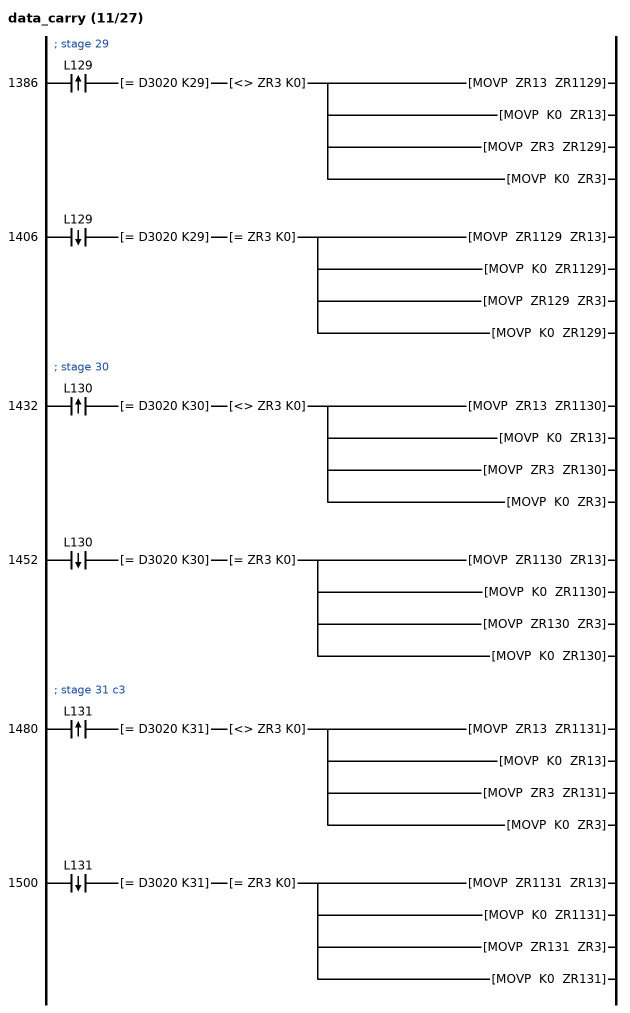
[picture p96: ladder of data_carry, rungs at steps 1386 to 1500]
; stage 29
1386  LDP     L129
      AND=    D3020 K29
      AND<>   ZR3 K0
      MOVP    ZR13 ZR1129
      MOVP    K0 ZR13
      MOVP    ZR3 ZR129
      MOVP    K0 ZR3
1406  LDF     L129
      AND=    D3020 K29
      AND=    ZR3 K0
      MOVP    ZR1129 ZR13
      MOVP    K0 ZR1129
      MOVP    ZR129 ZR3
      MOVP    K0 ZR129
; stage 30
1432  LDP     L130
      AND=    D3020 K30
      AND<>   ZR3 K0
      MOVP    ZR13 ZR1130
      MOVP    K0 ZR13
      MOVP    ZR3 ZR130
      MOVP    K0 ZR3
1452  LDF     L130
      AND=    D3020 K30
      AND=    ZR3 K0
      MOVP    ZR1130 ZR13
      MOVP    K0 ZR1130
      MOVP    ZR130 ZR3
      MOVP    K0 ZR130
; stage 31 c3
1480  LDP     L131
      AND=    D3020 K31
      AND<>   ZR3 K0
      MOVP    ZR13 ZR1131
      MOVP    K0 ZR13
      MOVP    ZR3 ZR131
      MOVP    K0 ZR3
1500  LDF     L131
      AND=    D3020 K31
      AND=    ZR3 K0
      MOVP    ZR1131 ZR13
      MOVP    K0 ZR1131
      MOVP    ZR131 ZR3
      MOVP    K0 ZR131
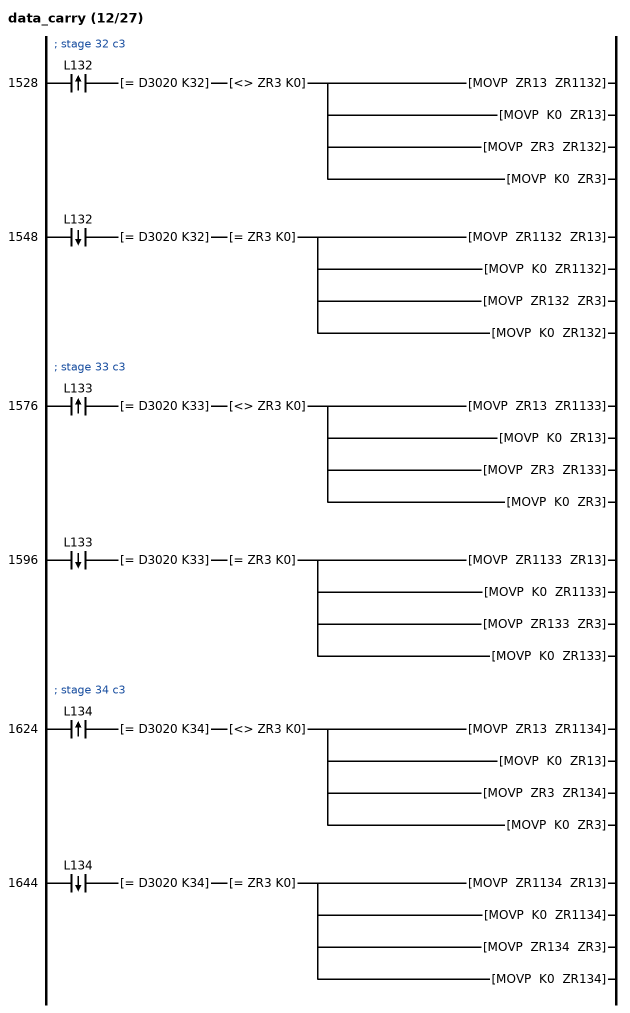
; stage 32 c3
1528  LDP     L132
      AND=    D3020 K32
      AND<>   ZR3 K0
      MOVP    ZR13 ZR1132
      MOVP    K0 ZR13
      MOVP    ZR3 ZR132
      MOVP    K0 ZR3
1548  LDF     L132
      AND=    D3020 K32
      AND=    ZR3 K0
      MOVP    ZR1132 ZR13
      MOVP    K0 ZR1132
      MOVP    ZR132 ZR3
      MOVP    K0 ZR132
; stage 33 c3
1576  LDP     L133
      AND=    D3020 K33
      AND<>   ZR3 K0
      MOVP    ZR13 ZR1133
      MOVP    K0 ZR13
      MOVP    ZR3 ZR133
      MOVP    K0 ZR3
1596  LDF     L133
      AND=    D3020 K33
      AND=    ZR3 K0
      MOVP    ZR1133 ZR13
      MOVP    K0 ZR1133
      MOVP    ZR133 ZR3
      MOVP    K0 ZR133
; stage 34 c3
1624  LDP     L134
      AND=    D3020 K34
      AND<>   ZR3 K0
      MOVP    ZR13 ZR1134
      MOVP    K0 ZR13
      MOVP    ZR3 ZR134
      MOVP    K0 ZR3
1644  LDF     L134
      AND=    D3020 K34
      AND=    ZR3 K0
      MOVP    ZR1134 ZR13
      MOVP    K0 ZR1134
      MOVP    ZR134 ZR3
      MOVP    K0 ZR134
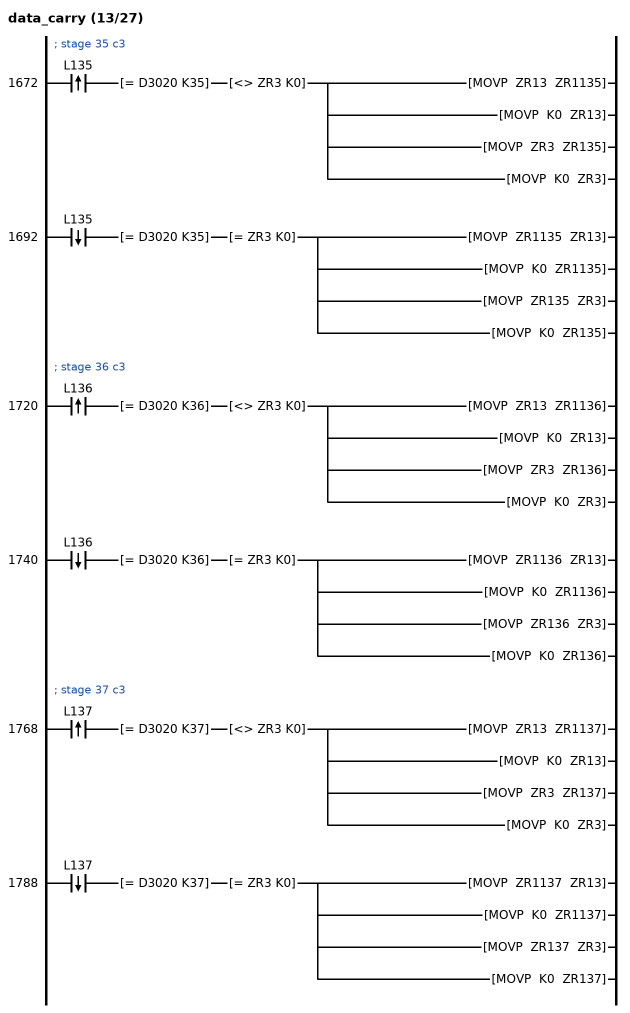
; stage 35 c3
1672  LDP     L135
      AND=    D3020 K35
      AND<>   ZR3 K0
      MOVP    ZR13 ZR1135
      MOVP    K0 ZR13
      MOVP    ZR3 ZR135
      MOVP    K0 ZR3
1692  LDF     L135
      AND=    D3020 K35
      AND=    ZR3 K0
      MOVP    ZR1135 ZR13
      MOVP    K0 ZR1135
      MOVP    ZR135 ZR3
      MOVP    K0 ZR135
; stage 36 c3
1720  LDP     L136
      AND=    D3020 K36
      AND<>   ZR3 K0
      MOVP    ZR13 ZR1136
      MOVP    K0 ZR13
      MOVP    ZR3 ZR136
      MOVP    K0 ZR3
1740  LDF     L136
      AND=    D3020 K36
      AND=    ZR3 K0
      MOVP    ZR1136 ZR13
      MOVP    K0 ZR1136
      MOVP    ZR136 ZR3
      MOVP    K0 ZR136
; stage 37 c3
1768  LDP     L137
      AND=    D3020 K37
      AND<>   ZR3 K0
      MOVP    ZR13 ZR1137
      MOVP    K0 ZR13
      MOVP    ZR3 ZR137
      MOVP    K0 ZR3
1788  LDF     L137
      AND=    D3020 K37
      AND=    ZR3 K0
      MOVP    ZR1137 ZR13
      MOVP    K0 ZR1137
      MOVP    ZR137 ZR3
      MOVP    K0 ZR137
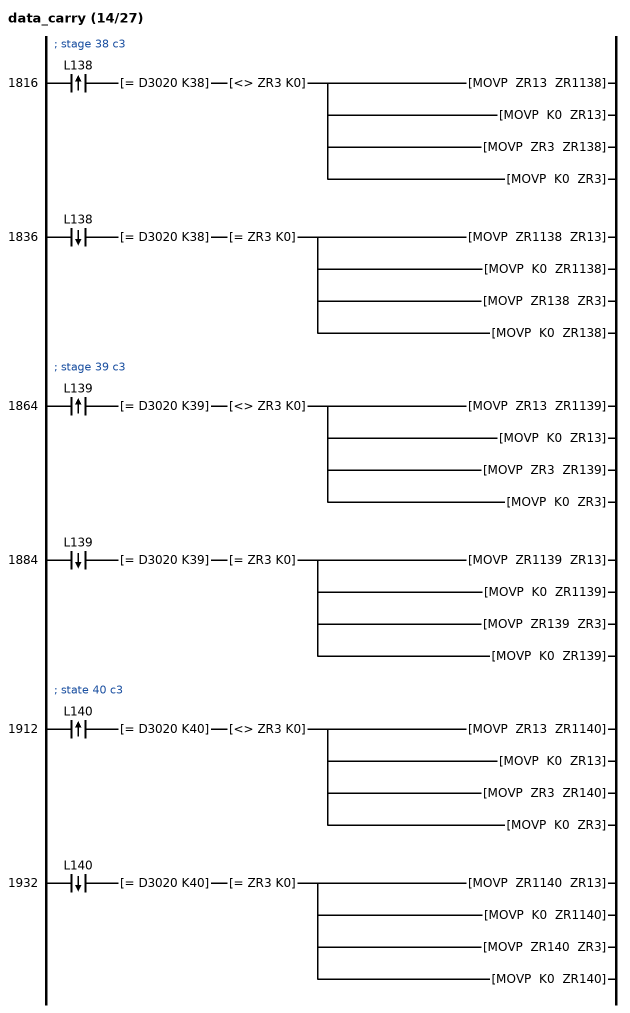
; stage 38 c3
1816  LDP     L138
      AND=    D3020 K38
      AND<>   ZR3 K0
      MOVP    ZR13 ZR1138
      MOVP    K0 ZR13
      MOVP    ZR3 ZR138
      MOVP    K0 ZR3
1836  LDF     L138
      AND=    D3020 K38
      AND=    ZR3 K0
      MOVP    ZR1138 ZR13
      MOVP    K0 ZR1138
      MOVP    ZR138 ZR3
      MOVP    K0 ZR138
; stage 39 c3
1864  LDP     L139
      AND=    D3020 K39
      AND<>   ZR3 K0
      MOVP    ZR13 ZR1139
      MOVP    K0 ZR13
      MOVP    ZR3 ZR139
      MOVP    K0 ZR3
1884  LDF     L139
      AND=    D3020 K39
      AND=    ZR3 K0
      MOVP    ZR1139 ZR13
      MOVP    K0 ZR1139
      MOVP    ZR139 ZR3
      MOVP    K0 ZR139
; state 40 c3
1912  LDP     L140
      AND=    D3020 K40
      AND<>   ZR3 K0
      MOVP    ZR13 ZR1140
      MOVP    K0 ZR13
      MOVP    ZR3 ZR140
      MOVP    K0 ZR3
1932  LDF     L140
      AND=    D3020 K40
      AND=    ZR3 K0
      MOVP    ZR1140 ZR13
      MOVP    K0 ZR1140
      MOVP    ZR140 ZR3
      MOVP    K0 ZR140
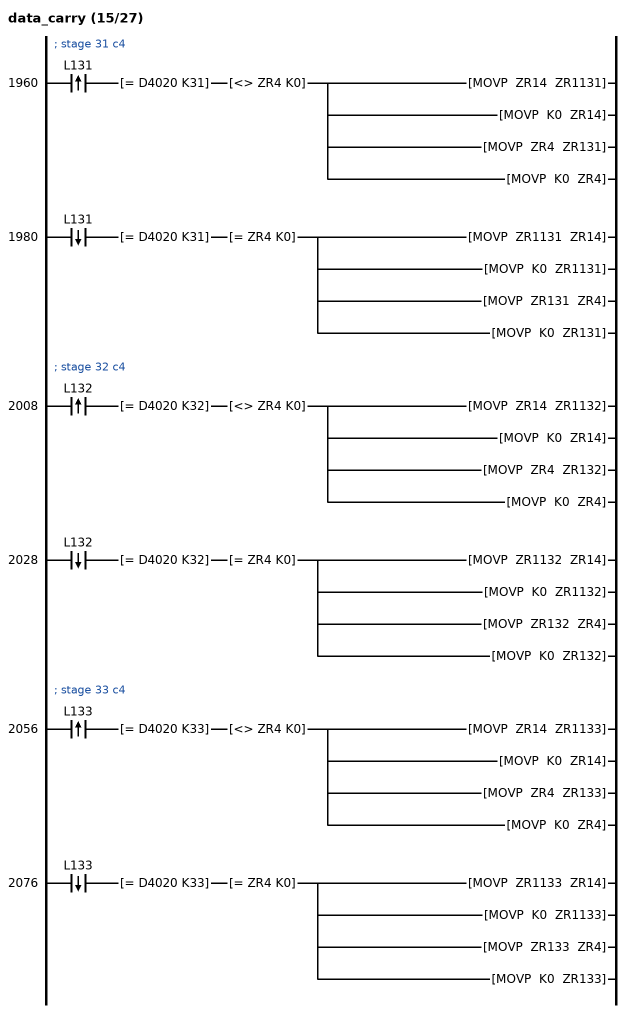
; stage 31 c4
1960  LDP     L131
      AND=    D4020 K31
      AND<>   ZR4 K0
      MOVP    ZR14 ZR1131
      MOVP    K0 ZR14
      MOVP    ZR4 ZR131
      MOVP    K0 ZR4
1980  LDF     L131
      AND=    D4020 K31
      AND=    ZR4 K0
      MOVP    ZR1131 ZR14
      MOVP    K0 ZR1131
      MOVP    ZR131 ZR4
      MOVP    K0 ZR131
; stage 32 c4
2008  LDP     L132
      AND=    D4020 K32
      AND<>   ZR4 K0
      MOVP    ZR14 ZR1132
      MOVP    K0 ZR14
      MOVP    ZR4 ZR132
      MOVP    K0 ZR4
2028  LDF     L132
      AND=    D4020 K32
      AND=    ZR4 K0
      MOVP    ZR1132 ZR14
      MOVP    K0 ZR1132
      MOVP    ZR132 ZR4
      MOVP    K0 ZR132
; stage 33 c4
2056  LDP     L133
      AND=    D4020 K33
      AND<>   ZR4 K0
      MOVP    ZR14 ZR1133
      MOVP    K0 ZR14
      MOVP    ZR4 ZR133
      MOVP    K0 ZR4
2076  LDF     L133
      AND=    D4020 K33
      AND=    ZR4 K0
      MOVP    ZR1133 ZR14
      MOVP    K0 ZR1133
      MOVP    ZR133 ZR4
      MOVP    K0 ZR133
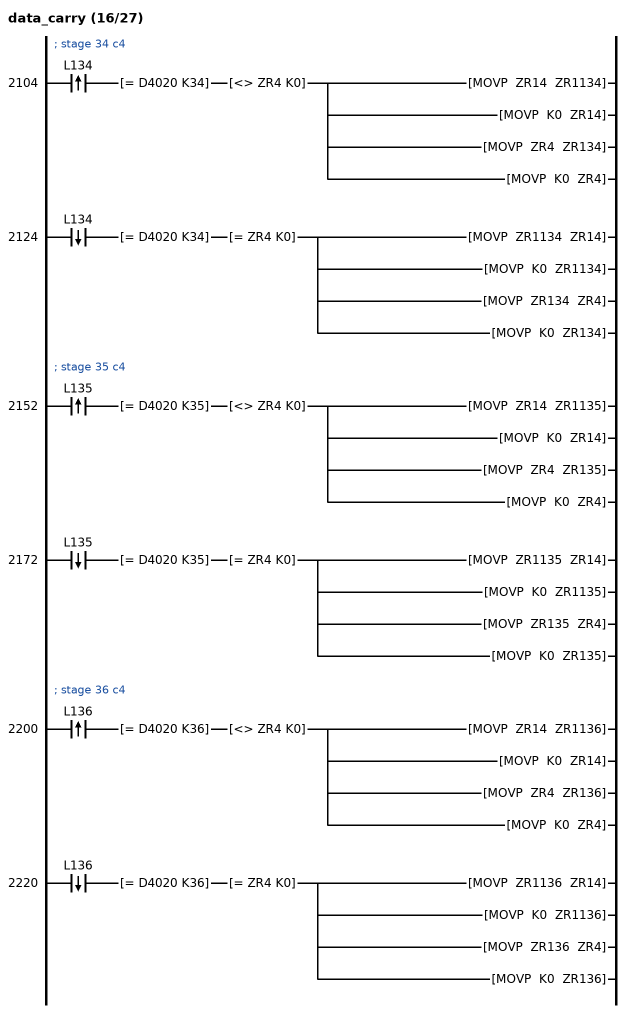
; stage 34 c4
2104  LDP     L134
      AND=    D4020 K34
      AND<>   ZR4 K0
      MOVP    ZR14 ZR1134
      MOVP    K0 ZR14
      MOVP    ZR4 ZR134
      MOVP    K0 ZR4
2124  LDF     L134
      AND=    D4020 K34
      AND=    ZR4 K0
      MOVP    ZR1134 ZR14
      MOVP    K0 ZR1134
      MOVP    ZR134 ZR4
      MOVP    K0 ZR134
; stage 35 c4
2152  LDP     L135
      AND=    D4020 K35
      AND<>   ZR4 K0
      MOVP    ZR14 ZR1135
      MOVP    K0 ZR14
      MOVP    ZR4 ZR135
      MOVP    K0 ZR4
2172  LDF     L135
      AND=    D4020 K35
      AND=    ZR4 K0
      MOVP    ZR1135 ZR14
      MOVP    K0 ZR1135
      MOVP    ZR135 ZR4
      MOVP    K0 ZR135
; stage 36 c4
2200  LDP     L136
      AND=    D4020 K36
      AND<>   ZR4 K0
      MOVP    ZR14 ZR1136
      MOVP    K0 ZR14
      MOVP    ZR4 ZR136
      MOVP    K0 ZR4
2220  LDF     L136
      AND=    D4020 K36
      AND=    ZR4 K0
      MOVP    ZR1136 ZR14
      MOVP    K0 ZR1136
      MOVP    ZR136 ZR4
      MOVP    K0 ZR136
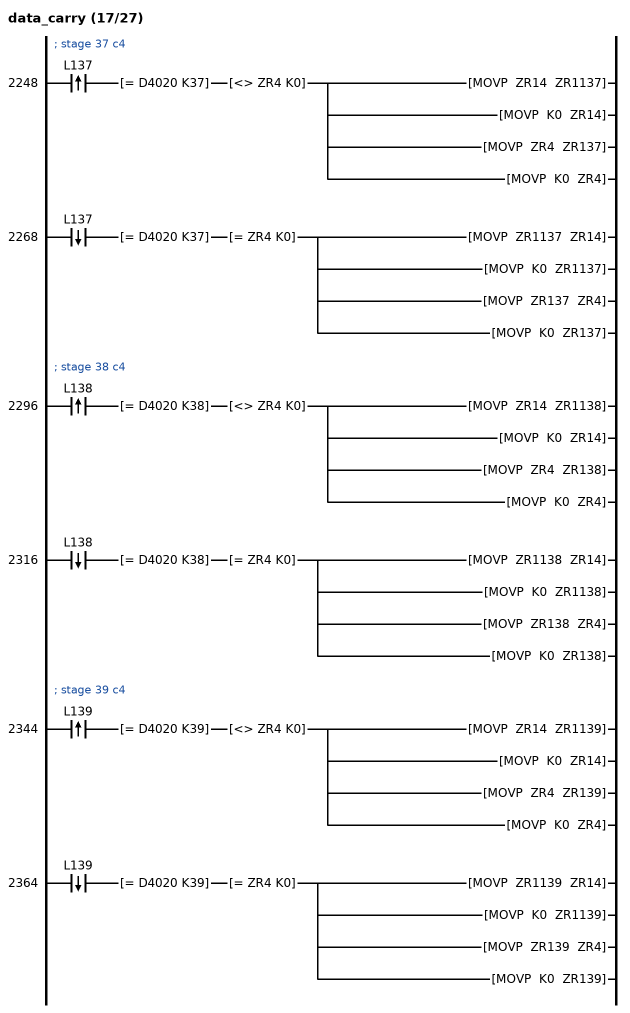
; stage 37 c4
2248  LDP     L137
      AND=    D4020 K37
      AND<>   ZR4 K0
      MOVP    ZR14 ZR1137
      MOVP    K0 ZR14
      MOVP    ZR4 ZR137
      MOVP    K0 ZR4
2268  LDF     L137
      AND=    D4020 K37
      AND=    ZR4 K0
      MOVP    ZR1137 ZR14
      MOVP    K0 ZR1137
      MOVP    ZR137 ZR4
      MOVP    K0 ZR137
; stage 38 c4
2296  LDP     L138
      AND=    D4020 K38
      AND<>   ZR4 K0
      MOVP    ZR14 ZR1138
      MOVP    K0 ZR14
      MOVP    ZR4 ZR138
      MOVP    K0 ZR4
2316  LDF     L138
      AND=    D4020 K38
      AND=    ZR4 K0
      MOVP    ZR1138 ZR14
      MOVP    K0 ZR1138
      MOVP    ZR138 ZR4
      MOVP    K0 ZR138
; stage 39 c4
2344  LDP     L139
      AND=    D4020 K39
      AND<>   ZR4 K0
      MOVP    ZR14 ZR1139
      MOVP    K0 ZR14
      MOVP    ZR4 ZR139
      MOVP    K0 ZR4
2364  LDF     L139
      AND=    D4020 K39
      AND=    ZR4 K0
      MOVP    ZR1139 ZR14
      MOVP    K0 ZR1139
      MOVP    ZR139 ZR4
      MOVP    K0 ZR139
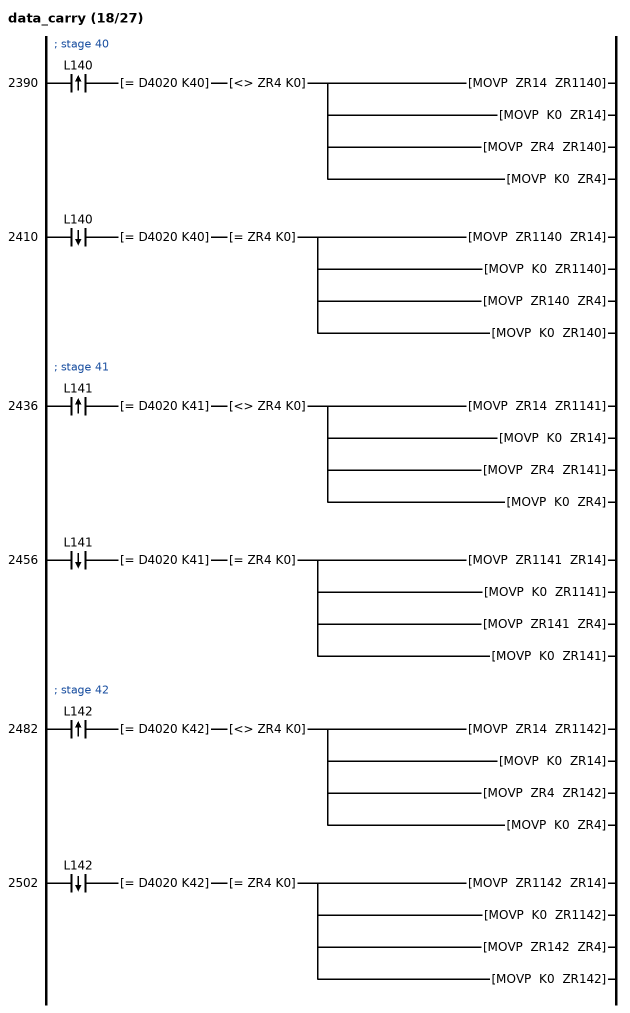
; stage 40
2390  LDP     L140
      AND=    D4020 K40
      AND<>   ZR4 K0
      MOVP    ZR14 ZR1140
      MOVP    K0 ZR14
      MOVP    ZR4 ZR140
      MOVP    K0 ZR4
2410  LDF     L140
      AND=    D4020 K40
      AND=    ZR4 K0
      MOVP    ZR1140 ZR14
      MOVP    K0 ZR1140
      MOVP    ZR140 ZR4
      MOVP    K0 ZR140
; stage 41
2436  LDP     L141
      AND=    D4020 K41
      AND<>   ZR4 K0
      MOVP    ZR14 ZR1141
      MOVP    K0 ZR14
      MOVP    ZR4 ZR141
      MOVP    K0 ZR4
2456  LDF     L141
      AND=    D4020 K41
      AND=    ZR4 K0
      MOVP    ZR1141 ZR14
      MOVP    K0 ZR1141
      MOVP    ZR141 ZR4
      MOVP    K0 ZR141
; stage 42
2482  LDP     L142
      AND=    D4020 K42
      AND<>   ZR4 K0
      MOVP    ZR14 ZR1142
      MOVP    K0 ZR14
      MOVP    ZR4 ZR142
      MOVP    K0 ZR4
2502  LDF     L142
      AND=    D4020 K42
      AND=    ZR4 K0
      MOVP    ZR1142 ZR14
      MOVP    K0 ZR1142
      MOVP    ZR142 ZR4
      MOVP    K0 ZR142
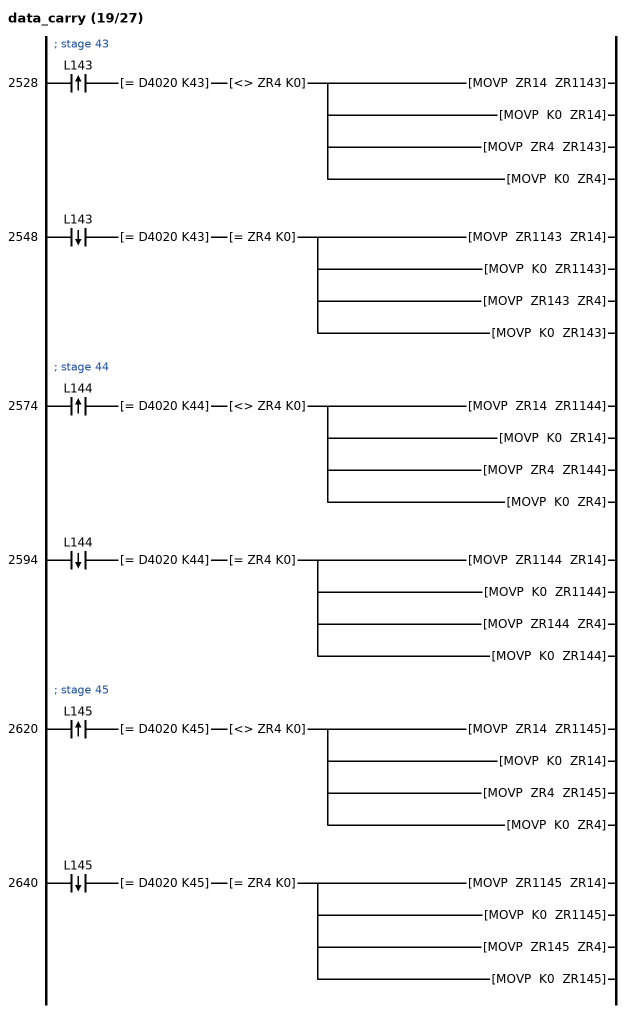
; stage 43
2528  LDP     L143
      AND=    D4020 K43
      AND<>   ZR4 K0
      MOVP    ZR14 ZR1143
      MOVP    K0 ZR14
      MOVP    ZR4 ZR143
      MOVP    K0 ZR4
2548  LDF     L143
      AND=    D4020 K43
      AND=    ZR4 K0
      MOVP    ZR1143 ZR14
      MOVP    K0 ZR1143
      MOVP    ZR143 ZR4
      MOVP    K0 ZR143
; stage 44
2574  LDP     L144
      AND=    D4020 K44
      AND<>   ZR4 K0
      MOVP    ZR14 ZR1144
      MOVP    K0 ZR14
      MOVP    ZR4 ZR144
      MOVP    K0 ZR4
2594  LDF     L144
      AND=    D4020 K44
      AND=    ZR4 K0
      MOVP    ZR1144 ZR14
      MOVP    K0 ZR1144
      MOVP    ZR144 ZR4
      MOVP    K0 ZR144
; stage 45
2620  LDP     L145
      AND=    D4020 K45
      AND<>   ZR4 K0
      MOVP    ZR14 ZR1145
      MOVP    K0 ZR14
      MOVP    ZR4 ZR145
      MOVP    K0 ZR4
2640  LDF     L145
      AND=    D4020 K45
      AND=    ZR4 K0
      MOVP    ZR1145 ZR14
      MOVP    K0 ZR1145
      MOVP    ZR145 ZR4
      MOVP    K0 ZR145
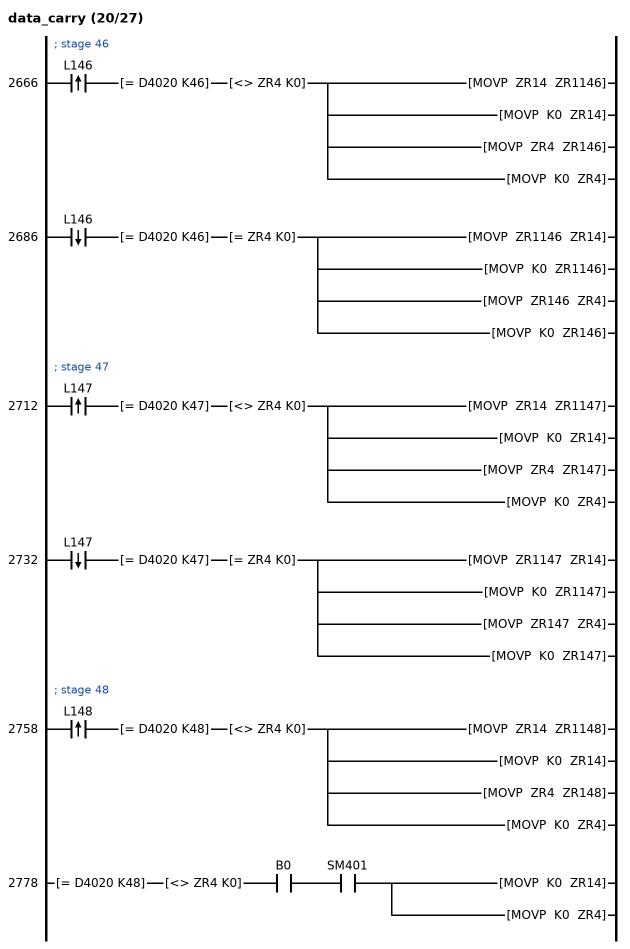
; stage 46
2666  LDP     L146
      AND=    D4020 K46
      AND<>   ZR4 K0
      MOVP    ZR14 ZR1146
      MOVP    K0 ZR14
      MOVP    ZR4 ZR146
      MOVP    K0 ZR4
2686  LDF     L146
      AND=    D4020 K46
      AND=    ZR4 K0
      MOVP    ZR1146 ZR14
      MOVP    K0 ZR1146
      MOVP    ZR146 ZR4
      MOVP    K0 ZR146
; stage 47
2712  LDP     L147
      AND=    D4020 K47
      AND<>   ZR4 K0
      MOVP    ZR14 ZR1147
      MOVP    K0 ZR14
      MOVP    ZR4 ZR147
      MOVP    K0 ZR4
2732  LDF     L147
      AND=    D4020 K47
      AND=    ZR4 K0
      MOVP    ZR1147 ZR14
      MOVP    K0 ZR1147
      MOVP    ZR147 ZR4
      MOVP    K0 ZR147
; stage 48
2758  LDP     L148
      AND=    D4020 K48
      AND<>   ZR4 K0
      MOVP    ZR14 ZR1148
      MOVP    K0 ZR14
      MOVP    ZR4 ZR148
      MOVP    K0 ZR4
2778  LD=     D4020 K48
      AND<>   ZR4 K0
      AND     B0
      AND     SM401
      MOVP    K0 ZR14
      MOVP    K0 ZR4
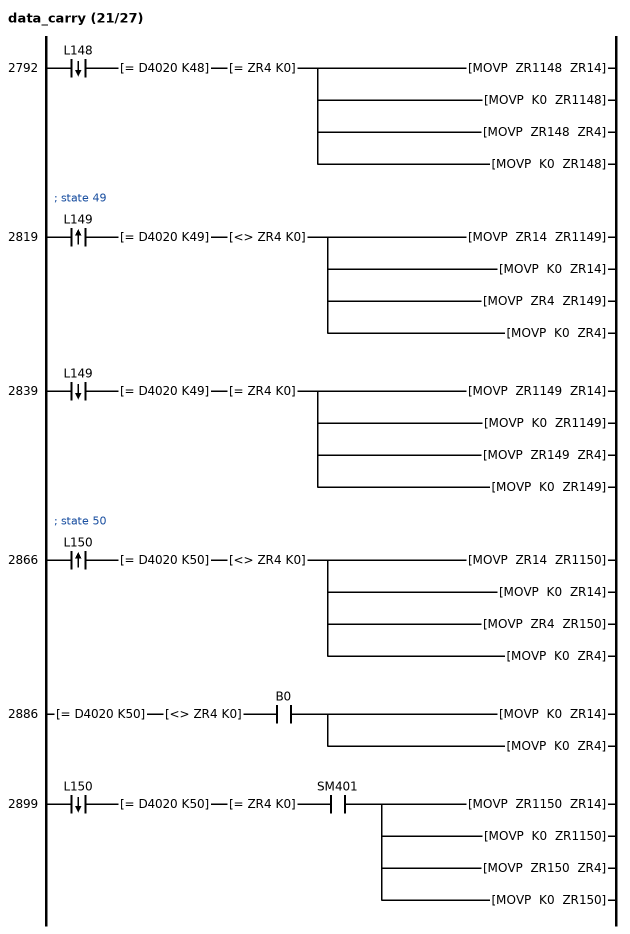
2792  LDF     L148
      AND=    D4020 K48
      AND=    ZR4 K0
      MOVP    ZR1148 ZR14
      MOVP    K0 ZR1148
      MOVP    ZR148 ZR4
      MOVP    K0 ZR148
; state 49
2819  LDP     L149
      AND=    D4020 K49
      AND<>   ZR4 K0
      MOVP    ZR14 ZR1149
      MOVP    K0 ZR14
      MOVP    ZR4 ZR149
      MOVP    K0 ZR4
2839  LDF     L149
      AND=    D4020 K49
      AND=    ZR4 K0
      MOVP    ZR1149 ZR14
      MOVP    K0 ZR1149
      MOVP    ZR149 ZR4
      MOVP    K0 ZR149
; state 50
2866  LDP     L150
      AND=    D4020 K50
      AND<>   ZR4 K0
      MOVP    ZR14 ZR1150
      MOVP    K0 ZR14
      MOVP    ZR4 ZR150
      MOVP    K0 ZR4
2886  LD=     D4020 K50
      AND<>   ZR4 K0
      AND     B0
      MOVP    K0 ZR14
      MOVP    K0 ZR4
2899  LDF     L150
      AND=    D4020 K50
      AND=    ZR4 K0
      AND     SM401
      MOVP    ZR1150 ZR14
      MOVP    K0 ZR1150
      MOVP    ZR150 ZR4
      MOVP    K0 ZR150
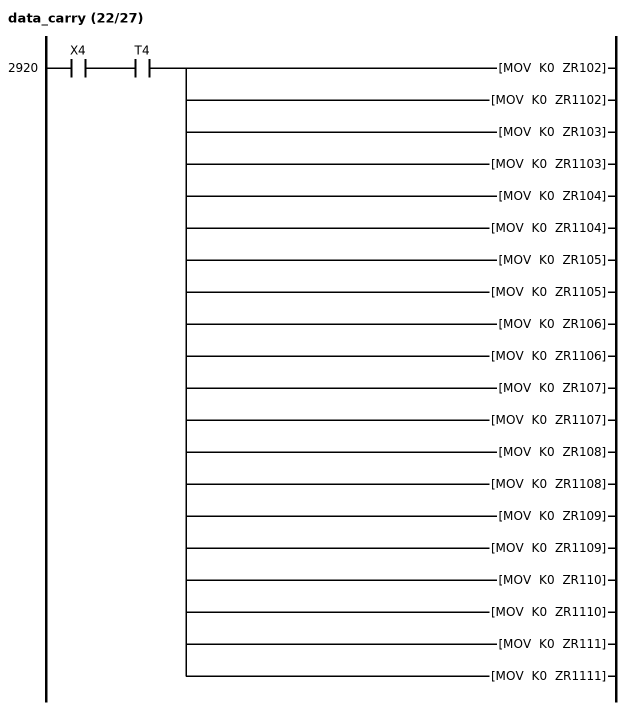
2920  LD      X4
      AND     T4
      MOV     K0 ZR102
      MOV     K0 ZR1102
      MOV     K0 ZR103
      MOV     K0 ZR1103
      MOV     K0 ZR104
      MOV     K0 ZR1104
      MOV     K0 ZR105
      MOV     K0 ZR1105
      MOV     K0 ZR106
      MOV     K0 ZR1106
      MOV     K0 ZR107
      MOV     K0 ZR1107
      MOV     K0 ZR108
      MOV     K0 ZR1108
      MOV     K0 ZR109
      MOV     K0 ZR1109
      MOV     K0 ZR110
      MOV     K0 ZR1110
      MOV     K0 ZR111
      MOV     K0 ZR1111
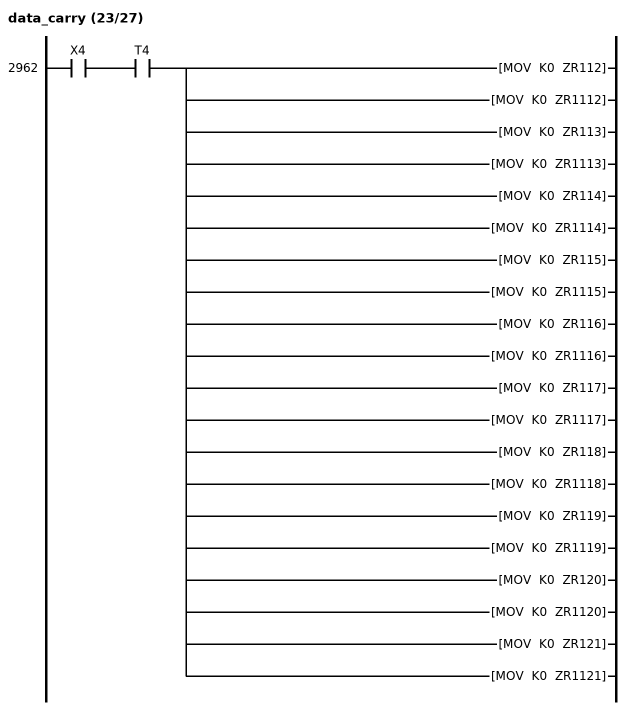
2962  LD      X4
      AND     T4
      MOV     K0 ZR112
      MOV     K0 ZR1112
      MOV     K0 ZR113
      MOV     K0 ZR1113
      MOV     K0 ZR114
      MOV     K0 ZR1114
      MOV     K0 ZR115
      MOV     K0 ZR1115
      MOV     K0 ZR116
      MOV     K0 ZR1116
      MOV     K0 ZR117
      MOV     K0 ZR1117
      MOV     K0 ZR118
      MOV     K0 ZR1118
      MOV     K0 ZR119
      MOV     K0 ZR1119
      MOV     K0 ZR120
      MOV     K0 ZR1120
      MOV     K0 ZR121
      MOV     K0 ZR1121
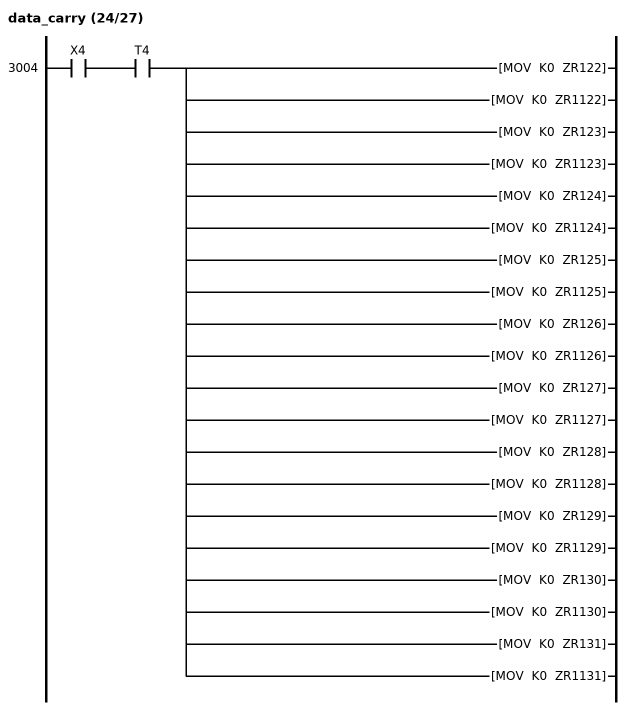
3004  LD      X4
      AND     T4
      MOV     K0 ZR122
      MOV     K0 ZR1122
      MOV     K0 ZR123
      MOV     K0 ZR1123
      MOV     K0 ZR124
      MOV     K0 ZR1124
      MOV     K0 ZR125
      MOV     K0 ZR1125
      MOV     K0 ZR126
      MOV     K0 ZR1126
      MOV     K0 ZR127
      MOV     K0 ZR1127
      MOV     K0 ZR128
      MOV     K0 ZR1128
      MOV     K0 ZR129
      MOV     K0 ZR1129
      MOV     K0 ZR130
      MOV     K0 ZR1130
      MOV     K0 ZR131
      MOV     K0 ZR1131
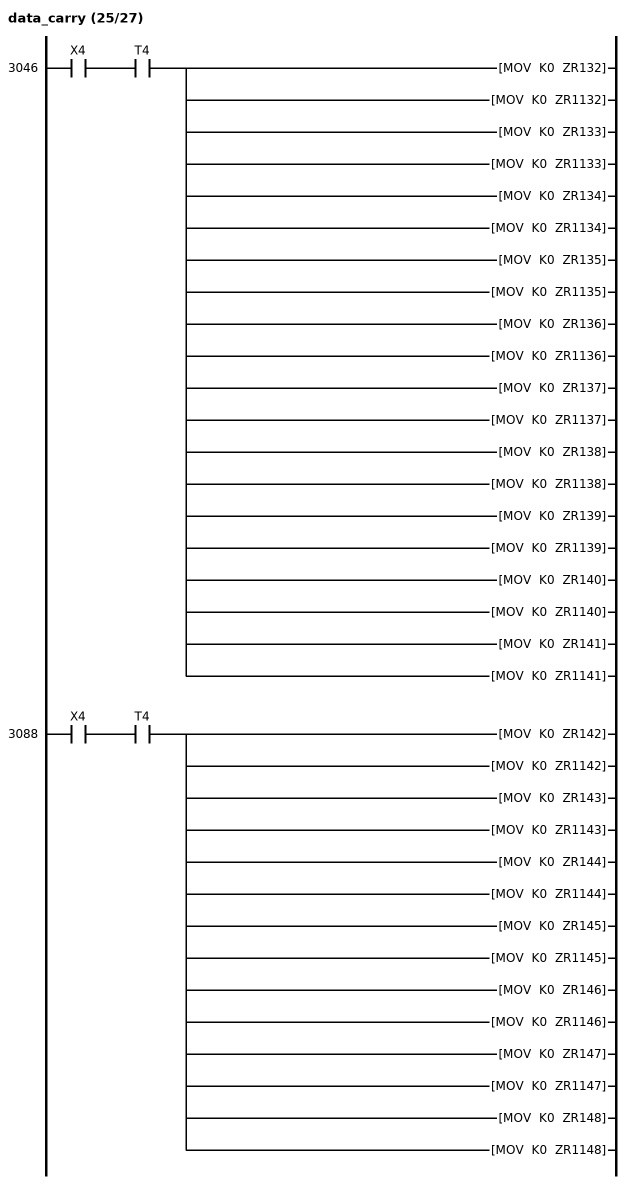
3046  LD      X4
      AND     T4
      MOV     K0 ZR132
      MOV     K0 ZR1132
      MOV     K0 ZR133
      MOV     K0 ZR1133
      MOV     K0 ZR134
      MOV     K0 ZR1134
      MOV     K0 ZR135
      MOV     K0 ZR1135
      MOV     K0 ZR136
      MOV     K0 ZR1136
      MOV     K0 ZR137
      MOV     K0 ZR1137
      MOV     K0 ZR138
      MOV     K0 ZR1138
      MOV     K0 ZR139
      MOV     K0 ZR1139
      MOV     K0 ZR140
      MOV     K0 ZR1140
      MOV     K0 ZR141
      MOV     K0 ZR1141
3088  LD      X4
      AND     T4
      MOV     K0 ZR142
      MOV     K0 ZR1142
      MOV     K0 ZR143
      MOV     K0 ZR1143
      MOV     K0 ZR144
      MOV     K0 ZR1144
      MOV     K0 ZR145
      MOV     K0 ZR1145
      MOV     K0 ZR146
      MOV     K0 ZR1146
      MOV     K0 ZR147
      MOV     K0 ZR1147
      MOV     K0 ZR148
      MOV     K0 ZR1148
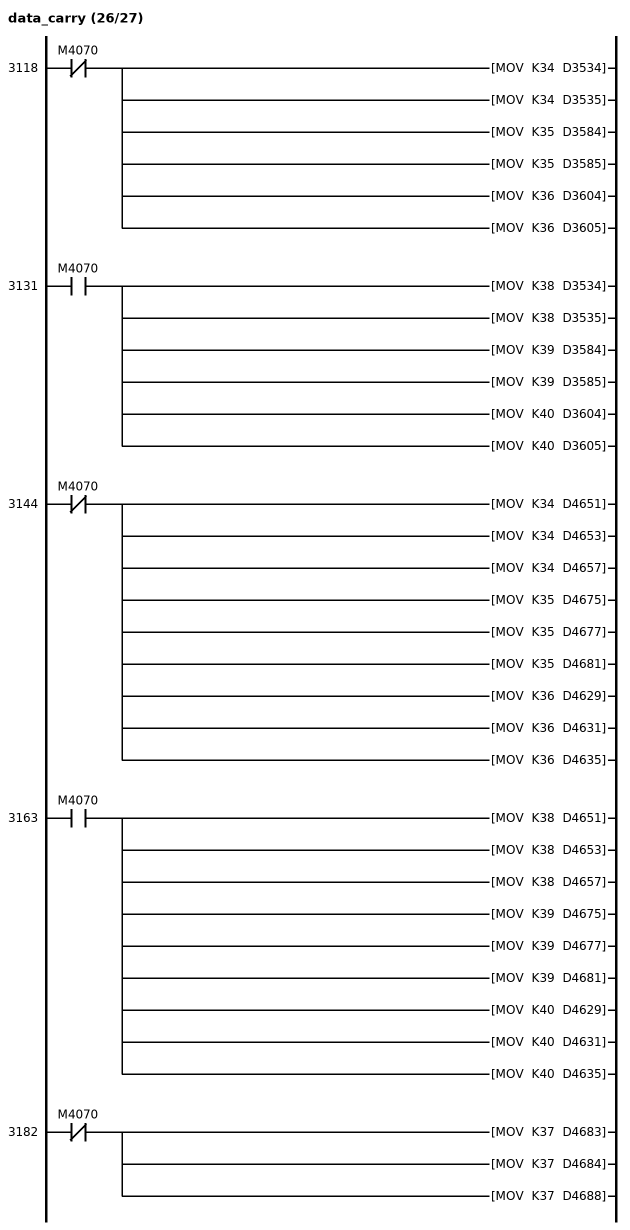
3118  LDI     M4070
      MOV     K34 D3534
      MOV     K34 D3535
      MOV     K35 D3584
      MOV     K35 D3585
      MOV     K36 D3604
      MOV     K36 D3605
3131  LD      M4070
      MOV     K38 D3534
      MOV     K38 D3535
      MOV     K39 D3584
      MOV     K39 D3585
      MOV     K40 D3604
      MOV     K40 D3605
3144  LDI     M4070
      MOV     K34 D4651
      MOV     K34 D4653
      MOV     K34 D4657
      MOV     K35 D4675
      MOV     K35 D4677
      MOV     K35 D4681
      MOV     K36 D4629
      MOV     K36 D4631
      MOV     K36 D4635
3163  LD      M4070
      MOV     K38 D4651
      MOV     K38 D4653
      MOV     K38 D4657
      MOV     K39 D4675
      MOV     K39 D4677
      MOV     K39 D4681
      MOV     K40 D4629
      MOV     K40 D4631
      MOV     K40 D4635
3182  LDI     M4070
      MOV     K37 D4683
      MOV     K37 D4684
      MOV     K37 D4688
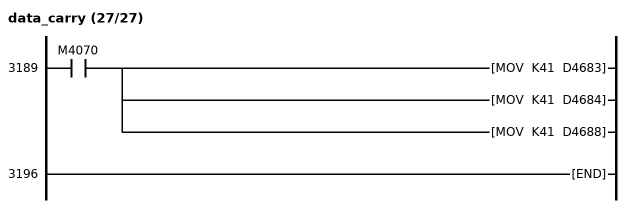
3189  LD      M4070
      MOV     K41 D4683
      MOV     K41 D4684
      MOV     K41 D4688
3196  END
END_PROGRAM

PROGRAM data_logger
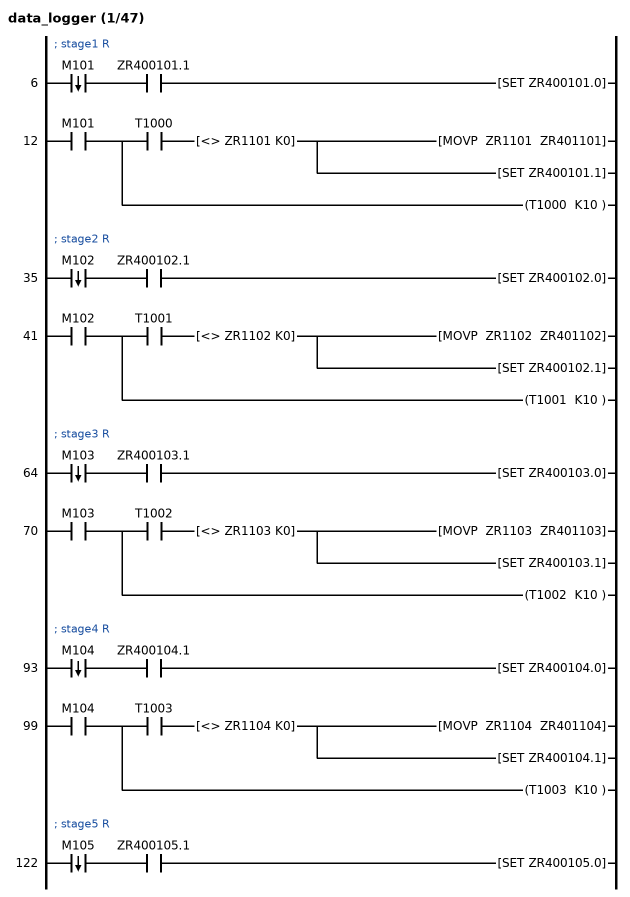
; stage1 R
6     LDF     M101
      AND     ZR400101.1
      SET     ZR400101.0
12    LD      M101
      MPS
      AND     T1000
      AND<>   ZR1101 K0
      MOVP    ZR1101 ZR401101
      SET     ZR400101.1
      MPP
      OUT     T1000 K10
; stage2 R
35    LDF     M102
      AND     ZR400102.1
      SET     ZR400102.0
41    LD      M102
      MPS
      AND     T1001
      AND<>   ZR1102 K0
      MOVP    ZR1102 ZR401102
      SET     ZR400102.1
      MPP
      OUT     T1001 K10
; stage3 R
64    LDF     M103
      AND     ZR400103.1
      SET     ZR400103.0
70    LD      M103
      MPS
      AND     T1002
      AND<>   ZR1103 K0
      MOVP    ZR1103 ZR401103
      SET     ZR400103.1
      MPP
      OUT     T1002 K10
; stage4 R
93    LDF     M104
      AND     ZR400104.1
      SET     ZR400104.0
99    LD      M104
      MPS
      AND     T1003
      AND<>   ZR1104 K0
      MOVP    ZR1104 ZR401104
      SET     ZR400104.1
      MPP
      OUT     T1003 K10
; stage5 R
122   LDF     M105
      AND     ZR400105.1
      SET     ZR400105.0
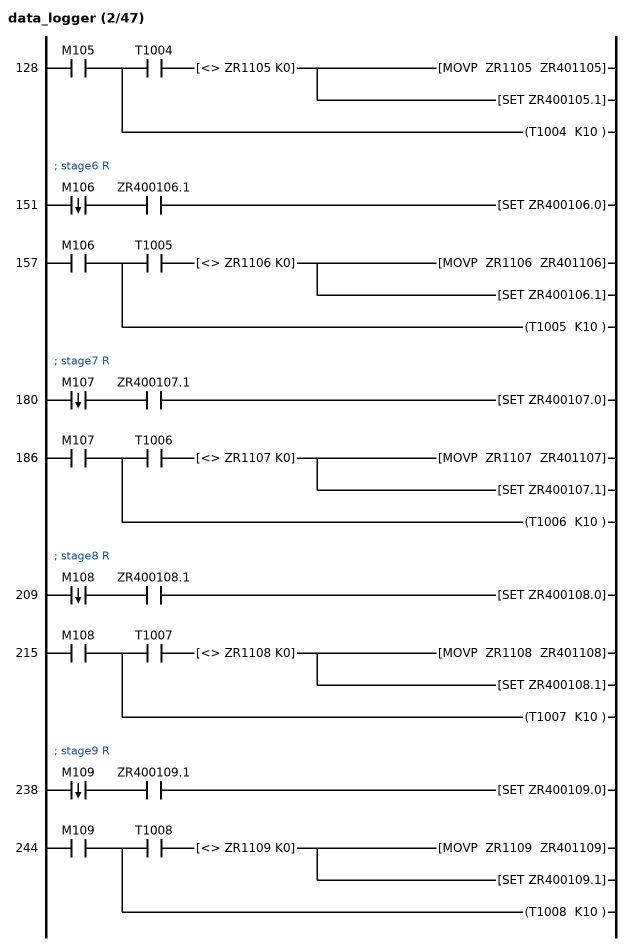
128   LD      M105
      MPS
      AND     T1004
      AND<>   ZR1105 K0
      MOVP    ZR1105 ZR401105
      SET     ZR400105.1
      MPP
      OUT     T1004 K10
; stage6 R
151   LDF     M106
      AND     ZR400106.1
      SET     ZR400106.0
157   LD      M106
      MPS
      AND     T1005
      AND<>   ZR1106 K0
      MOVP    ZR1106 ZR401106
      SET     ZR400106.1
      MPP
      OUT     T1005 K10
; stage7 R
180   LDF     M107
      AND     ZR400107.1
      SET     ZR400107.0
186   LD      M107
      MPS
      AND     T1006
      AND<>   ZR1107 K0
      MOVP    ZR1107 ZR401107
      SET     ZR400107.1
      MPP
      OUT     T1006 K10
; stage8 R
209   LDF     M108
      AND     ZR400108.1
      SET     ZR400108.0
215   LD      M108
      MPS
      AND     T1007
      AND<>   ZR1108 K0
      MOVP    ZR1108 ZR401108
      SET     ZR400108.1
      MPP
      OUT     T1007 K10
; stage9 R
238   LDF     M109
      AND     ZR400109.1
      SET     ZR400109.0
244   LD      M109
      MPS
      AND     T1008
      AND<>   ZR1109 K0
      MOVP    ZR1109 ZR401109
      SET     ZR400109.1
      MPP
      OUT     T1008 K10
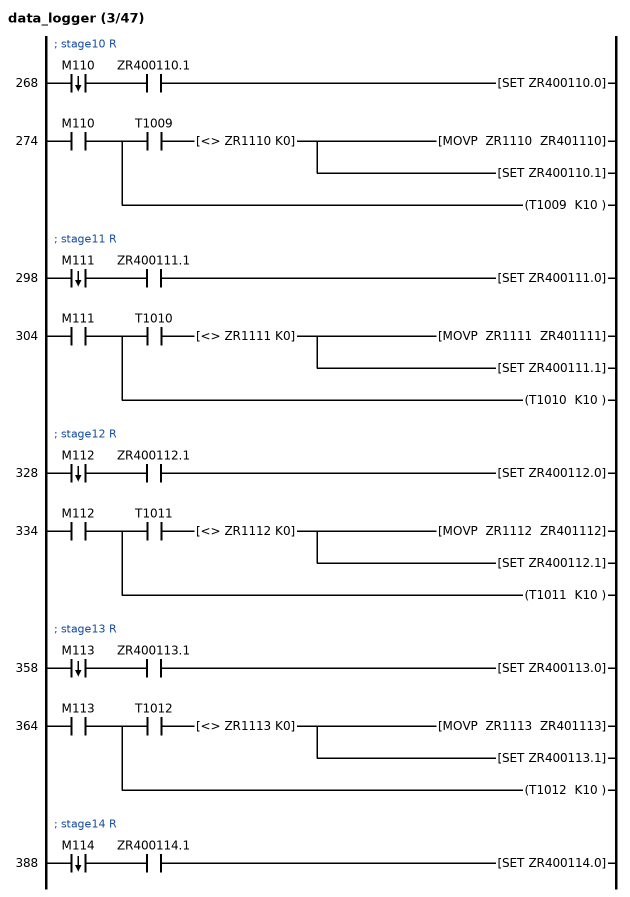
; stage10 R
268   LDF     M110
      AND     ZR400110.1
      SET     ZR400110.0
274   LD      M110
      MPS
      AND     T1009
      AND<>   ZR1110 K0
      MOVP    ZR1110 ZR401110
      SET     ZR400110.1
      MPP
      OUT     T1009 K10
; stage11 R
298   LDF     M111
      AND     ZR400111.1
      SET     ZR400111.0
304   LD      M111
      MPS
      AND     T1010
      AND<>   ZR1111 K0
      MOVP    ZR1111 ZR401111
      SET     ZR400111.1
      MPP
      OUT     T1010 K10
; stage12 R
328   LDF     M112
      AND     ZR400112.1
      SET     ZR400112.0
334   LD      M112
      MPS
      AND     T1011
      AND<>   ZR1112 K0
      MOVP    ZR1112 ZR401112
      SET     ZR400112.1
      MPP
      OUT     T1011 K10
; stage13 R
358   LDF     M113
      AND     ZR400113.1
      SET     ZR400113.0
364   LD      M113
      MPS
      AND     T1012
      AND<>   ZR1113 K0
      MOVP    ZR1113 ZR401113
      SET     ZR400113.1
      MPP
      OUT     T1012 K10
; stage14 R
388   LDF     M114
      AND     ZR400114.1
      SET     ZR400114.0
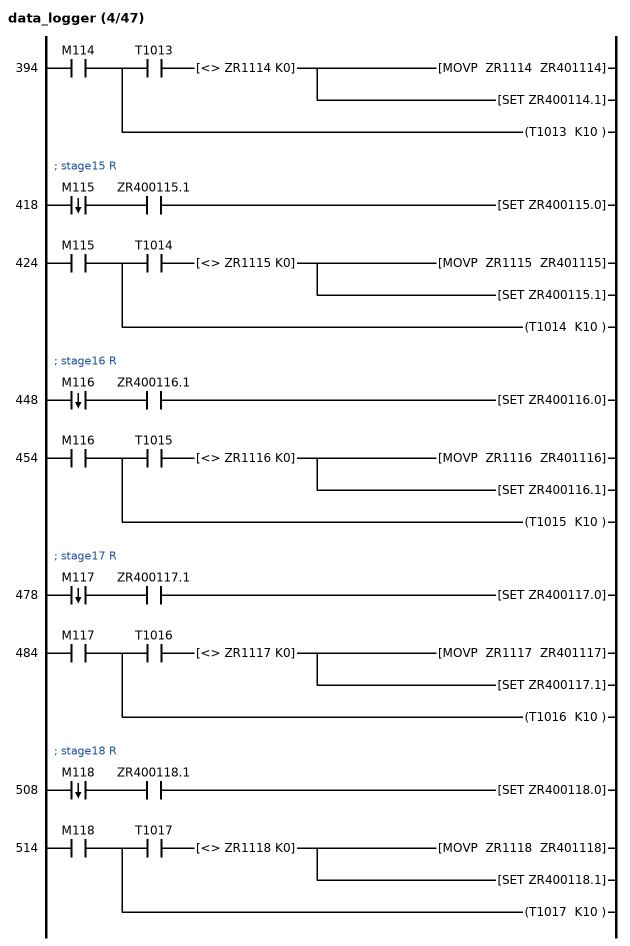
394   LD      M114
      MPS
      AND     T1013
      AND<>   ZR1114 K0
      MOVP    ZR1114 ZR401114
      SET     ZR400114.1
      MPP
      OUT     T1013 K10
; stage15 R
418   LDF     M115
      AND     ZR400115.1
      SET     ZR400115.0
424   LD      M115
      MPS
      AND     T1014
      AND<>   ZR1115 K0
      MOVP    ZR1115 ZR401115
      SET     ZR400115.1
      MPP
      OUT     T1014 K10
; stage16 R
448   LDF     M116
      AND     ZR400116.1
      SET     ZR400116.0
454   LD      M116
      MPS
      AND     T1015
      AND<>   ZR1116 K0
      MOVP    ZR1116 ZR401116
      SET     ZR400116.1
      MPP
      OUT     T1015 K10
; stage17 R
478   LDF     M117
      AND     ZR400117.1
      SET     ZR400117.0
484   LD      M117
      MPS
      AND     T1016
      AND<>   ZR1117 K0
      MOVP    ZR1117 ZR401117
      SET     ZR400117.1
      MPP
      OUT     T1016 K10
; stage18 R
508   LDF     M118
      AND     ZR400118.1
      SET     ZR400118.0
514   LD      M118
      MPS
      AND     T1017
      AND<>   ZR1118 K0
      MOVP    ZR1118 ZR401118
      SET     ZR400118.1
      MPP
      OUT     T1017 K10
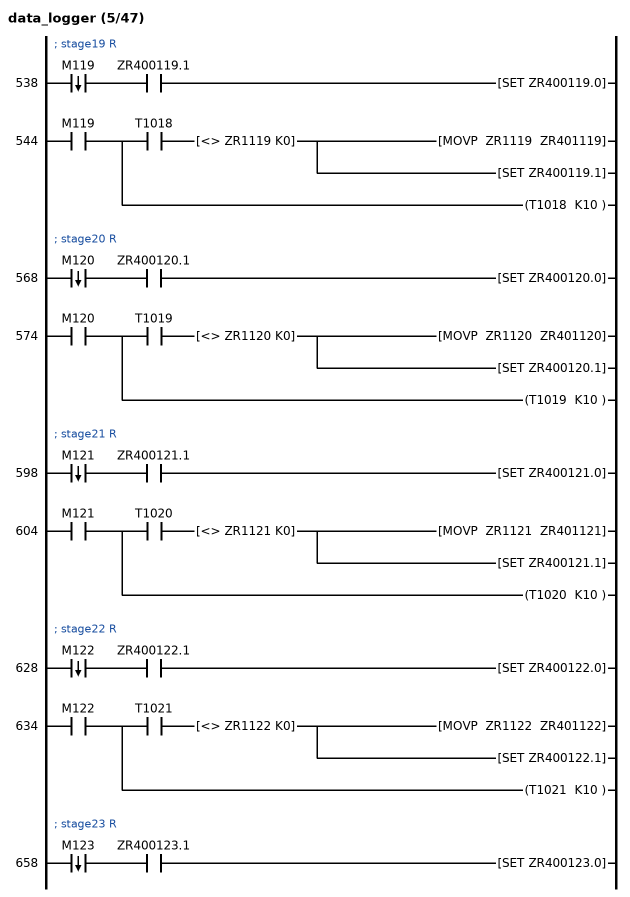
; stage19 R
538   LDF     M119
      AND     ZR400119.1
      SET     ZR400119.0
544   LD      M119
      MPS
      AND     T1018
      AND<>   ZR1119 K0
      MOVP    ZR1119 ZR401119
      SET     ZR400119.1
      MPP
      OUT     T1018 K10
; stage20 R
568   LDF     M120
      AND     ZR400120.1
      SET     ZR400120.0
574   LD      M120
      MPS
      AND     T1019
      AND<>   ZR1120 K0
      MOVP    ZR1120 ZR401120
      SET     ZR400120.1
      MPP
      OUT     T1019 K10
; stage21 R
598   LDF     M121
      AND     ZR400121.1
      SET     ZR400121.0
604   LD      M121
      MPS
      AND     T1020
      AND<>   ZR1121 K0
      MOVP    ZR1121 ZR401121
      SET     ZR400121.1
      MPP
      OUT     T1020 K10
; stage22 R
628   LDF     M122
      AND     ZR400122.1
      SET     ZR400122.0
634   LD      M122
      MPS
      AND     T1021
      AND<>   ZR1122 K0
      MOVP    ZR1122 ZR401122
      SET     ZR400122.1
      MPP
      OUT     T1021 K10
; stage23 R
658   LDF     M123
      AND     ZR400123.1
      SET     ZR400123.0
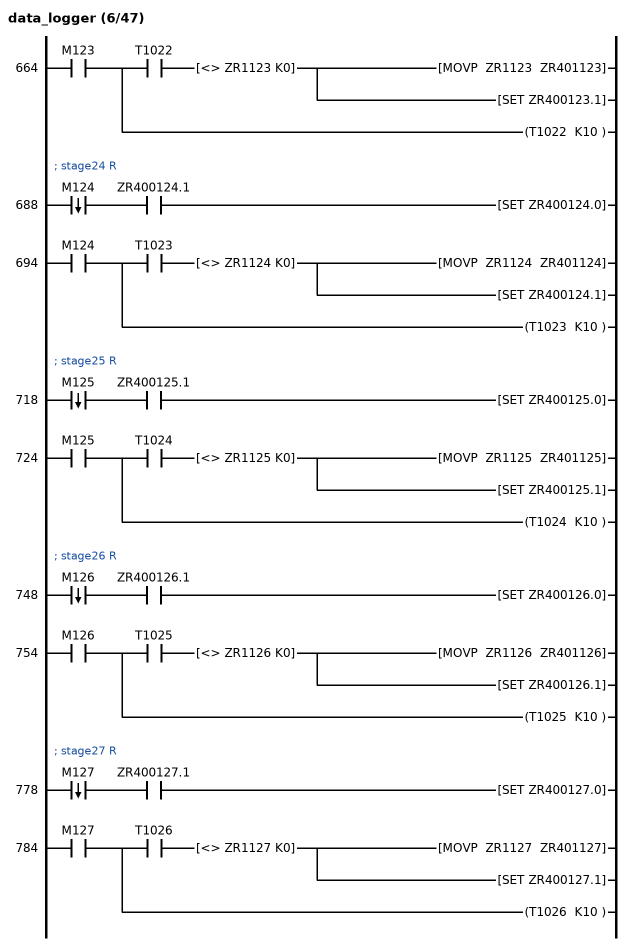
664   LD      M123
      MPS
      AND     T1022
      AND<>   ZR1123 K0
      MOVP    ZR1123 ZR401123
      SET     ZR400123.1
      MPP
      OUT     T1022 K10
; stage24 R
688   LDF     M124
      AND     ZR400124.1
      SET     ZR400124.0
694   LD      M124
      MPS
      AND     T1023
      AND<>   ZR1124 K0
      MOVP    ZR1124 ZR401124
      SET     ZR400124.1
      MPP
      OUT     T1023 K10
; stage25 R
718   LDF     M125
      AND     ZR400125.1
      SET     ZR400125.0
724   LD      M125
      MPS
      AND     T1024
      AND<>   ZR1125 K0
      MOVP    ZR1125 ZR401125
      SET     ZR400125.1
      MPP
      OUT     T1024 K10
; stage26 R
748   LDF     M126
      AND     ZR400126.1
      SET     ZR400126.0
754   LD      M126
      MPS
      AND     T1025
      AND<>   ZR1126 K0
      MOVP    ZR1126 ZR401126
      SET     ZR400126.1
      MPP
      OUT     T1025 K10
; stage27 R
778   LDF     M127
      AND     ZR400127.1
      SET     ZR400127.0
784   LD      M127
      MPS
      AND     T1026
      AND<>   ZR1127 K0
      MOVP    ZR1127 ZR401127
      SET     ZR400127.1
      MPP
      OUT     T1026 K10
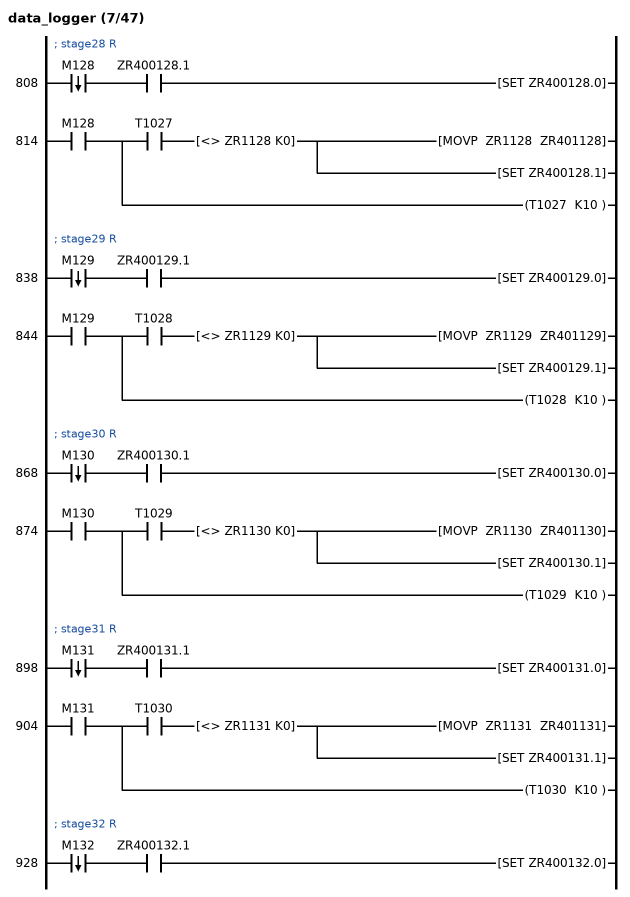
; stage28 R
808   LDF     M128
      AND     ZR400128.1
      SET     ZR400128.0
814   LD      M128
      MPS
      AND     T1027
      AND<>   ZR1128 K0
      MOVP    ZR1128 ZR401128
      SET     ZR400128.1
      MPP
      OUT     T1027 K10
; stage29 R
838   LDF     M129
      AND     ZR400129.1
      SET     ZR400129.0
844   LD      M129
      MPS
      AND     T1028
      AND<>   ZR1129 K0
      MOVP    ZR1129 ZR401129
      SET     ZR400129.1
      MPP
      OUT     T1028 K10
; stage30 R
868   LDF     M130
      AND     ZR400130.1
      SET     ZR400130.0
874   LD      M130
      MPS
      AND     T1029
      AND<>   ZR1130 K0
      MOVP    ZR1130 ZR401130
      SET     ZR400130.1
      MPP
      OUT     T1029 K10
; stage31 R
898   LDF     M131
      AND     ZR400131.1
      SET     ZR400131.0
904   LD      M131
      MPS
      AND     T1030
      AND<>   ZR1131 K0
      MOVP    ZR1131 ZR401131
      SET     ZR400131.1
      MPP
      OUT     T1030 K10
; stage32 R
928   LDF     M132
      AND     ZR400132.1
      SET     ZR400132.0
